(* PLC project workshop_4, Desconocido Sin nombre 1 *)
(* stored: creationDateTime 2024-03-30T18:45:35, modificationDateTime 2024-04-01T02:17:35 *)

PROGRAM workshop_4
  VAR
    B1 AT %IX0.0 : BOOL;
    B2 AT %IX0.1 : BOOL;
    B3 AT %IX0.2 : BOOL;
    H1 AT %QX0.0 : BOOL;
    H2 AT %QX0.1 : BOOL;
    H3 AT %QX0.2 : BOOL;
    H4 AT %QX0.3 : BOOL;
    H5 AT %QX0.4 : BOOL;
  END_VAR

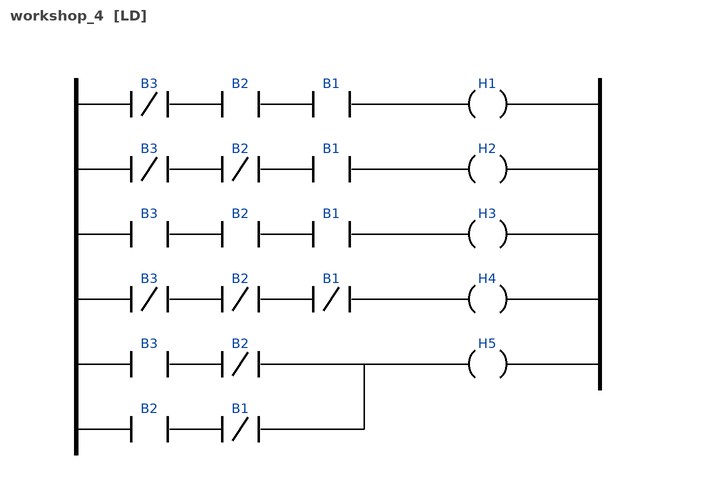
(* LD diagram, written out as Structured Text *)
H1 := NOT B3 AND B2 AND B1;
H2 := NOT B3 AND NOT B2 AND B1;
H3 := B3 AND B2 AND B1;
H4 := NOT B3 AND NOT B2 AND NOT B1;
H5 := B3 AND NOT B2 OR B2 AND NOT B1;
END_PROGRAM

CONFIGURATION Config0
  RESOURCE Res0 ON PLC
    TASK task0(INTERVAL := T#20ms, PRIORITY := 0);
    PROGRAM instance0 WITH task0 : workshop_4;
  END_RESOURCE
END_CONFIGURATION
